TYPE E_Room :
(
	Hall := 0,
	Kitchen := 1,
	BedRoom1 := 2,
	BedRoom2 := 3
);
END_TYPE

(* stored: Version 1.1.0.1, ProductVersion 3.1.4024.13
   DUT E_Room: Id {fac28bca-530a-44d9-878c-72a8b23f1226} *)
